Yaskawa INFORM job: MAKE-UF.JBI

/JOB
//NAME MAKE-UF
///FOLDERNAME FOLDER001
//POS
///NPOS 2,0,0,0,0,0
///TOOL 1
///POSTYPE PULSE
///PULSE
C00000=-652,-17775,21844,-416,-82513,491
C00001=-361,56948,97542,-215,-89436,245
//INST
///DATE 2025/09/30 15:12
///ATTR SC,RW
///GROUP1 RB1
///LVARS 0,0,10,0,0,0,0,0
NOP
SFTOF
PAUSE
MOVL C00000 V=166.7  //ORG
MOVL C00001 V=166.7  //XX
END
